Universal Robots PolyScope program: test1.urp

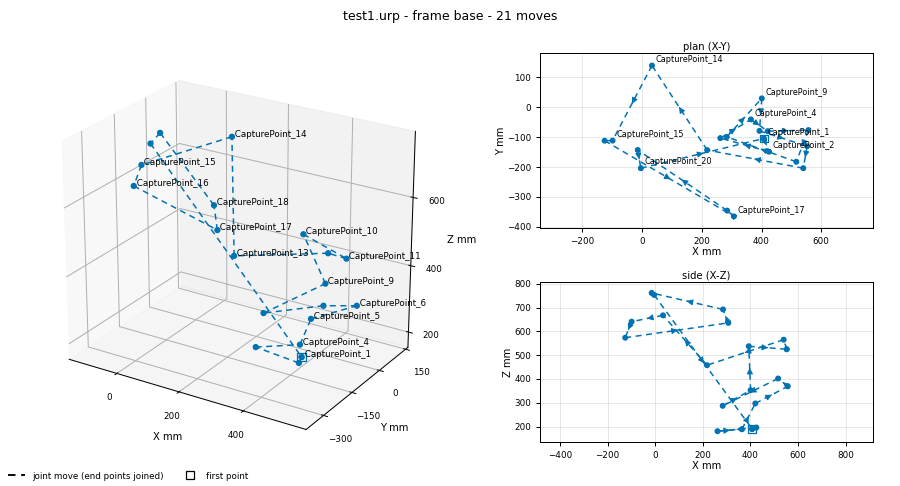
[picture p0: tool path of test1.urp in frame base, 21 of 21 moves have a stored position in this frame; points joined in program order, loops and branches not executed]
Program test1 (installation=default directory=/programs createdIn=3.8.0.61336 lastSavedIn=3.8.0.61336 robotSerialNumber=2016352774)
Calibrated DH parameters: a=[0.000165, -0.326475, -0.363587, -0.000196, 0.000314, 0]; d=[0.089242, 611.192012, -553.715229, -57.366527, 0.094858, 0.082351]; alpha=[1.570545, 0.000446, 0.002569, 1.569839, -1.569769, 0]; deltaTheta=[-0.000028, 0.695517, -0.309849, -0.385645, -0.000052, -0.000026]
Robot Program (runOnlyOnce=false)
  Script file /programs/X0.script
    | address="172.16.58.34"
    | port=3000
    | sname="mt"
    | socket_open(address,port,sname)
    | p=get_actual_tcp_pose()
    | socket_send_line("X0()",sname)
    | ret=socket_read_line(sname)
    | socket_close(sname)
  MoveJ speed 60 deg/s, acceleration 80 deg/s^2 (useActiveTCP=false)
    Waypoint CapturePoint_1: TCP in base x=407.319 y=-104.477 z=189.798 mm, rx=0.0132 ry=-3.0834 rz=0.0275 rad; joints [1.102, -90.323, -126.824, -56.254, 89.174, 0.603] deg; flange x=407.369 y=-104.477 z=189.795 mm, rx=2.1925 ry=-2.1741 rz=-0.0439 rad
  Wait Sleep waitTime=1
  Script file /programs/X1.script
    | address="172.16.58.34"
    | port=3000
    | timeout=10
    | socket_open(address,port)
    | p=get_actual_tcp_pose()
    | rpy=rotvec2rpy([p[3],p[4],p[5]])
    | socket_send_string("X1(")
    | socket_send_string(p[0])
    | socket_send_string(",")
    | socket_send_string(p[1])
    | socket_send_string(",")
    | socket_send_string(p[2])
    | socket_send_string(",")
    | socket_send_string(r2d(rpy[0]))
    | socket_send_string(",")
    | socket_send_string(r2d(rpy[1]))
    | socket_send_string(",")
    | socket_send_string(r2d(rpy[2]))
    | socket_send_line(")")
    | ret=socket_read_line(timeout=10)
    | if (ret!="OK"):
    |   code=socket_read_string()
    |   popup(code,title="X1",blocking=True)
    | end
    | socket_close()
  MoveJ speed 60 deg/s, acceleration 80 deg/s^2 (useActiveTCP=false)
    Waypoint CapturePoint_2: TCP in base x=425.113 y=-148.666 z=195.791 mm, rx=-0.1792 ry=-3.0783 rz=-0.2322 rad; joints [-6.597, -94.285, -121.705, -57.418, 98.578, -0.232] deg
  Wait Sleep waitTime=1
  Script file /programs/X1.script
    | address="172.16.58.34"
    | port=3000
    | timeout=10
    | socket_open(address,port)
    | p=get_actual_tcp_pose()
    | rpy=rotvec2rpy([p[3],p[4],p[5]])
    | socket_send_string("X1(")
    | socket_send_string(p[0])
    | socket_send_string(",")
    | socket_send_string(p[1])
    | socket_send_string(",")
    | socket_send_string(p[2])
    | socket_send_string(",")
    | socket_send_string(r2d(rpy[0]))
    | socket_send_string(",")
    | socket_send_string(r2d(rpy[1]))
    | socket_send_string(",")
    | socket_send_string(r2d(rpy[2]))
    | socket_send_line(")")
    | ret=socket_read_line(timeout=10)
    | socket_close()
    | popup(ret,title="X1",blocking=True)
  MoveJ speed 60 deg/s, acceleration 80 deg/s^2 (useActiveTCP=false)
    Waypoint CapturePoint_3: TCP in base x=261.868 y=-103.158 z=180.589 mm, rx=0.0437 ry=2.8124 rz=-0.0205 rad; joints [2.246, -68.558, -152.367, -30.363, 88.291, 3.753] deg; flange x=261.915 y=-103.159 z=180.605 mm, rx=-2.0171 ry=2.081 rz=-0.355 rad
  Wait Sleep waitTime=1
  Script file /programs/X1.script
    | (same text as the earlier copy of this file)
  Wait Sleep waitTime=1
  MoveJ speed 60 deg/s, acceleration 80 deg/s^2 (useActiveTCP=false)
    Waypoint CapturePoint_4: TCP in base x=364.401 y=-40.427 z=188.676 mm, rx=-0.0839 ry=3.0452 rz=-0.4018 rad; joints [14.918, -81.577, -136.612, -51.472, 74.61, 11.698] deg; flange x=364.451 y=-40.423 z=188.679 mm, rx=2.1677 ry=-2.0517 rz=0.3517 rad
  Wait Sleep waitTime=1
  Script file /programs/X1.script
    | (same text as the earlier copy of this file)
  MoveJ speed 60 deg/s, acceleration 80 deg/s^2 (useActiveTCP=false)
    Waypoint CapturePoint_5: TCP in base x=420.711 y=-79.895 z=297.199 mm, rx=-1.2251 ry=-2.8429 rz=0.1199 rad; joints [4.807, -83.549, -115.101, -75.705, 87.411, 51.451] deg; flange x=420.746 y=-79.931 z=297.198 mm, rx=1.1291 ry=-2.8395 rz=0.0366 rad
  Wait Sleep waitTime=1
  Script file /programs/X1.script
    | (same text as the earlier copy of this file)
  MoveJ speed 60 deg/s, acceleration 80 deg/s^2 (useActiveTCP=false)
    Waypoint CapturePoint_6: TCP in base x=557.015 y=-76.212 z=369.049 mm, rx=-1.1202 ry=-2.6042 rz=0.326 rad; joints [4.185, -103.414, -80.018, -107.33, 86.262, 51.278] deg
  Wait Sleep waitTime=1
  Script file /programs/X1.script
    | (same text as the earlier copy of this file)
  MoveJ speed 60 deg/s, acceleration 80 deg/s^2 (useActiveTCP=false)
    Waypoint CapturePoint_7: TCP in base x=516.519 y=-182.473 z=401.871 mm, rx=-0.4638 ry=-2.819 rz=-0.3213 rad; joints [-9.651, -100.545, -79.796, -105.39, 102.635, 7.132] deg; flange x=516.565 y=-182.487 z=401.857 mm, rx=1.7858 ry=-2.4894 rz=-0.536 rad
  Wait Sleep waitTime=1
  Script file /programs/X1.script
    | (same text as the earlier copy of this file)
  MoveJ speed 60 deg/s, acceleration 80 deg/s^2 (useActiveTCP=false)
    Waypoint CapturePoint_8: TCP in base x=283.57 y=-98.864 z=287.1 mm, rx=0.1306 ry=2.9178 rz=-0.0523 rad; joints [3.423, -60.53, -136.111, -61.056, 86.82, 8.151] deg
  Wait Sleep waitTime=1
  Script file /programs/X1.script
    | (same text as the earlier copy of this file)
  MoveJ speed 60 deg/s, acceleration 80 deg/s^2 (useActiveTCP=false)
    Waypoint CapturePoint_9: TCP in base x=400.864 y=30.008 z=352.811 mm, rx=0.0271 ry=-3.0726 rz=0.5533 rad; joints [24.159, -77.716, -110.963, -90.885, 71.963, 24.568] deg; flange x=400.914 y=30.009 z=352.81 mm, rx=2.037 ry=-2.0016 rz=0.3436 rad
  Wait Sleep waitTime=1
  Script file /programs/X1.script
    | (same text as the earlier copy of this file)
  MoveJ speed 60 deg/s, acceleration 80 deg/s^2 (useActiveTCP=false)
    Waypoint CapturePoint_10: TCP in base x=393.15 y=-78.817 z=537.403 mm, rx=-0.3142 ry=-3.0516 rz=0.0028 rad; joints [4.609, -79.583, -82.759, -111.9, 90.771, 16.175] deg
  Wait Sleep waitTime=1
  Script file /programs/X1.script
    | (same text as the earlier copy of this file)
  MoveJ speed 60 deg/s, acceleration 80 deg/s^2 (useActiveTCP=false)
    Waypoint CapturePoint_11: TCP in base x=552.83 y=-130.286 z=524.726 mm, rx=-0.4744 ry=-2.8257 rz=0.0233 rad; joints [-2.134, -106.285, -53.992, -125.607, 91.185, 16.575] deg; flange x=552.875 y=-130.302 z=524.713 mm, rx=1.6958 ry=-2.3803 rz=-0.2705 rad
  Wait Sleep waitTime=1
  Script file /programs/X1.script
    | (same text as the earlier copy of this file)
  MoveJ speed 60 deg/s, acceleration 80 deg/s^2 (useActiveTCP=false)
    Waypoint CapturePoint_12: TCP in base x=539.794 y=-203.877 z=565.039 mm, rx=-1.1778 ry=-2.608 rz=-0.1105 rad; joints [-10.728, -110.456, -42.192, -131.984, 97.99, 36.654] deg; flange x=539.826 y=-203.913 z=565.025 mm, rx=1.0515 ry=-2.7841 rz=-0.3757 rad
  Wait Sleep waitTime=1
  Script file /programs/X1.script
    | (same text as the earlier copy of this file)
  MoveJ speed 60 deg/s, acceleration 80 deg/s^2 (useActiveTCP=false)
    Waypoint CapturePoint_13: TCP in base x=217.74 y=-143.133 z=457.721 mm, rx=1.04 ry=2.7655 rz=0.2418 rad; joints [-10.661, -53.703, -113.544, -91.144, 97.517, 31.19] deg; flange x=217.777 y=-143.166 z=457.726 mm, rx=-1.1979 ry=2.6421 rz=-0.0149 rad
  Wait Sleep waitTime=1
  Script file /programs/X1.script
    | (same text as the earlier copy of this file)
  Halt
  MoveJ speed 60 deg/s, acceleration 80 deg/s^2 (useActiveTCP=false)
    Waypoint CapturePoint_14: TCP in base x=32.955 y=140.061 z=667.229 mm, rx=-1.0077 ry=2.5472 rz=-0.74 rad; joints [-127.955, -38.755, -66.496, -163.608, 124.335, -79.153] deg
  Wait Sleep waitTime=1
  Script file /programs/X1.script
    | (same text as the earlier copy of this file)
  MoveJ speed 60 deg/s, acceleration 80 deg/s^2 (useActiveTCP=false)
    Waypoint CapturePoint_15: TCP in base x=-98.976 y=-111.429 z=640.718 mm, rx=-1.9221 ry=1.7558 rz=-0.7168 rad; joints [0.392, -27.054, -85.502, -117.851, 86.877, -4.56] deg
  Wait Sleep waitTime=1
  Script file /programs/X1.script
    | (same text as the earlier copy of this file)
  MoveJ speed 60 deg/s, acceleration 80 deg/s^2 (useActiveTCP=false)
    Waypoint CapturePoint_16: TCP in base x=-125.724 y=-111.715 z=573.266 mm, rx=-1.7134 ry=1.786 rz=-0.7532 rad; joints [0.402, -15.524, -97.784, -110.625, 86.851, 2.752] deg
  Wait Sleep waitTime=1
  Script file /programs/X1.script
    | (same text as the earlier copy of this file)
  MoveJ speed 60 deg/s, acceleration 80 deg/s^2 (useActiveTCP=false)
    Waypoint CapturePoint_17: TCP in base x=307.338 y=-365.217 z=635.603 mm, rx=-1.8392 ry=1.9097 rz=0.7596 rad; joints [-40.903, -107.911, -31.186, -161.588, 113.228, -43.898] deg
  Wait Sleep waitTime=1
  Script file /programs/X1.script
    | (same text as the earlier copy of this file)
  MoveJ speed 60 deg/s, acceleration 80 deg/s^2 (useActiveTCP=false)
    Waypoint CapturePoint_18: TCP in base x=285.042 y=-346.037 z=692.112 mm, rx=-0.2019 ry=-2.9931 rz=-0.8493 rad; joints [-40.903, -107.916, -21.263, -161.588, 113.234, 53.855] deg
  Wait Sleep waitTime=1
  Script file /programs/X1.script
    | (same text as the earlier copy of this file)
  MoveJ speed 60 deg/s, acceleration 80 deg/s^2 (useActiveTCP=false)
    Waypoint CapturePoint_19: TCP in base x=-14.788 y=-142.877 z=761.304 mm, rx=0.9846 ry=2.4689 rz=0.6334 rad; joints [-71.114, -70.355, -47.356, -156.575, 124.411, 62.513] deg
  Wait Sleep waitTime=1
  Script file /programs/X1.script
    | (same text as the earlier copy of this file)
  MoveJ speed 60 deg/s, acceleration 80 deg/s^2 (useActiveTCP=false)
    Waypoint CapturePoint_20: TCP in base x=-4.371 y=-203.918 z=753.086 mm, rx=-1.8631 ry=1.8783 rz=-0.0962 rad; joints [-71.114, -77.335, -43.394, -157.914, 116.465, -71.239] deg
  Wait Sleep waitTime=1
  Script file /programs/X1.script
    | (same text as the earlier copy of this file)
  MoveJ speed 60 deg/s, acceleration 80 deg/s^2 (useActiveTCP=false)
    Waypoint CapturePoint_1: TCP in base x=407.319 y=-104.477 z=189.798 mm, rx=0.0132 ry=-3.0834 rz=0.0275 rad; joints [1.102, -90.323, -126.824, -56.254, 89.174, 0.603] deg; flange x=407.369 y=-104.477 z=189.795 mm, rx=2.1925 ry=-2.1741 rz=-0.0439 rad
  Halt
